FUNCTION_BLOCK FB_AnimalController
VAR_INPUT
END_VAR
VAR_OUTPUT
END_VAR
VAR
	ipGetAnimal: I_AnimalTraits;
END_VAR

END_FUNCTION_BLOCK

(* stored: Version 1.1.0.1, ProductVersion 3.1.4024.16
   POU FB_AnimalController: Id {8b4655ac-5146-4060-8aa2-52ed6ed809fc}, SpecialFunc None *)
